INTERFACE I_PidController

METHOD AutomaticControl : BOOL
VAR_INPUT
	processVariable		: REAL; // Temperature measurement
	setpoint			: REAL; // Temperature setpoint
END_VAR
END_METHOD

METHOD ManualControl : BOOL
VAR_INPUT
	iControlPercentage : INT;
END_VAR
END_METHOD

METHOD ResetControl : BOOL
END_METHOD

METHOD SetParameters : BOOL
VAR_INPUT
	parameters			: ST_PidParameters;
END_VAR
END_METHOD

END_INTERFACE

(* stored: Version 1.1.0.1, ProductVersion 3.1.4024.9
   Itf I_PidController: Id {aa630658-0d8b-4e8d-a461-2fcb82cd964a}
   Method AutomaticControl: Id {faea0406-8ebf-41f1-9459-a5ac78b7e924}
   Method ManualControl: Id {04f20102-d226-4c81-b17e-1d3eaeea885c}
   Method ResetControl: Id {0357bd7b-59ca-496b-a283-938b826645e7}
   Method SetParameters: Id {c9bcb76f-994e-4fce-8534-5f8b44dc3dbe} *)
